TYPE ST_UCDevices :
STRUCT
	Status : ST_UC_Status;
END_STRUCT
END_TYPE

(* stored: Version 1.1.0.1, ProductVersion 3.1.4024.11
   DUT ST_UCDevices: Id {72f99cea-875d-4cc9-8e63-b57e51b8d303} *)
